(* CODESYS project BagFeeder.xml

Project tree, tasks and I/O mapping:
  function block BagFeeder [CFC]
*)

// BagFeeder
FUNCTION_BLOCK BagFeeder
//  .					.					.
VAR_INPUT
	BagOpenSensor: BOOL;
	IceFullSensor: BOOL;
	HeatSealOpened: BOOL;
	HeatSealClosed: BOOL;
	CheckBagOpenDelay: TIME;
	RetryBagOpenDelay: TIME;
	MaxIceFeedTime: TIME;
	IceTopOffTime: TIME;
	SealingTime: TIME;
	HeatSealCompleteDelay: TIME;
	//BagOpenRetries: UINT;
	
	BaggerSettings: BaggerSettings;
	
	Trigger: BOOL;
	MotionComplete: BOOL;
	
END_VAR
VAR_OUTPUT
	BlowerOn: BOOL;
	FillIce: BOOL;
	OpenHeatSeal: BOOL;
	CloseHeatSeal: BOOL;
	BagOpenRetryAttempts: UINT;
	
	ExecuteMotion: BOOL;
	MotionSteps: UDINT;
	MotionDirection: UINT;
	MotionSpeed: UINT;
	MotionTriggerOnSensor: BOOL;
END_VAR
VAR
	_MakeBagSequence: MakeBagSequence;
	_BagAdvanceSequence: BagAdvanceSequence; 
	_FeedIceSequence: FeedIceSequence;
	_SealBagSequence: SealBagSequence;
	
	_FailOpenCounter: CTU;
	_ResetFailCounter: BOOL;
	
	_MotionSelector: MotionSelector;
	
	_TestBagAdvance: BOOL;
	_TestFirstAdvance: BOOL;
	_TestFirstRetract: BOOL;
	_TestRetryAdvance: BOOL;
	_TestRetryRetract: BOOL;
	_TestTearBag: BOOL;
	_TestResetBag: BOOL;
	_TestRetractOneBag: BOOL;
	_TestBlowerOn: BOOL;
	MotionCompleteTrigger: R_TRIG;
	_TestHeatSeal: BOOL;
END_VAR
VAR // added by the converter: edge detectors and wires of the graphical bodies
    _w1, _w2, _w3, _w4, _w5, _w6, _w7, _w8 : ANY;
END_VAR

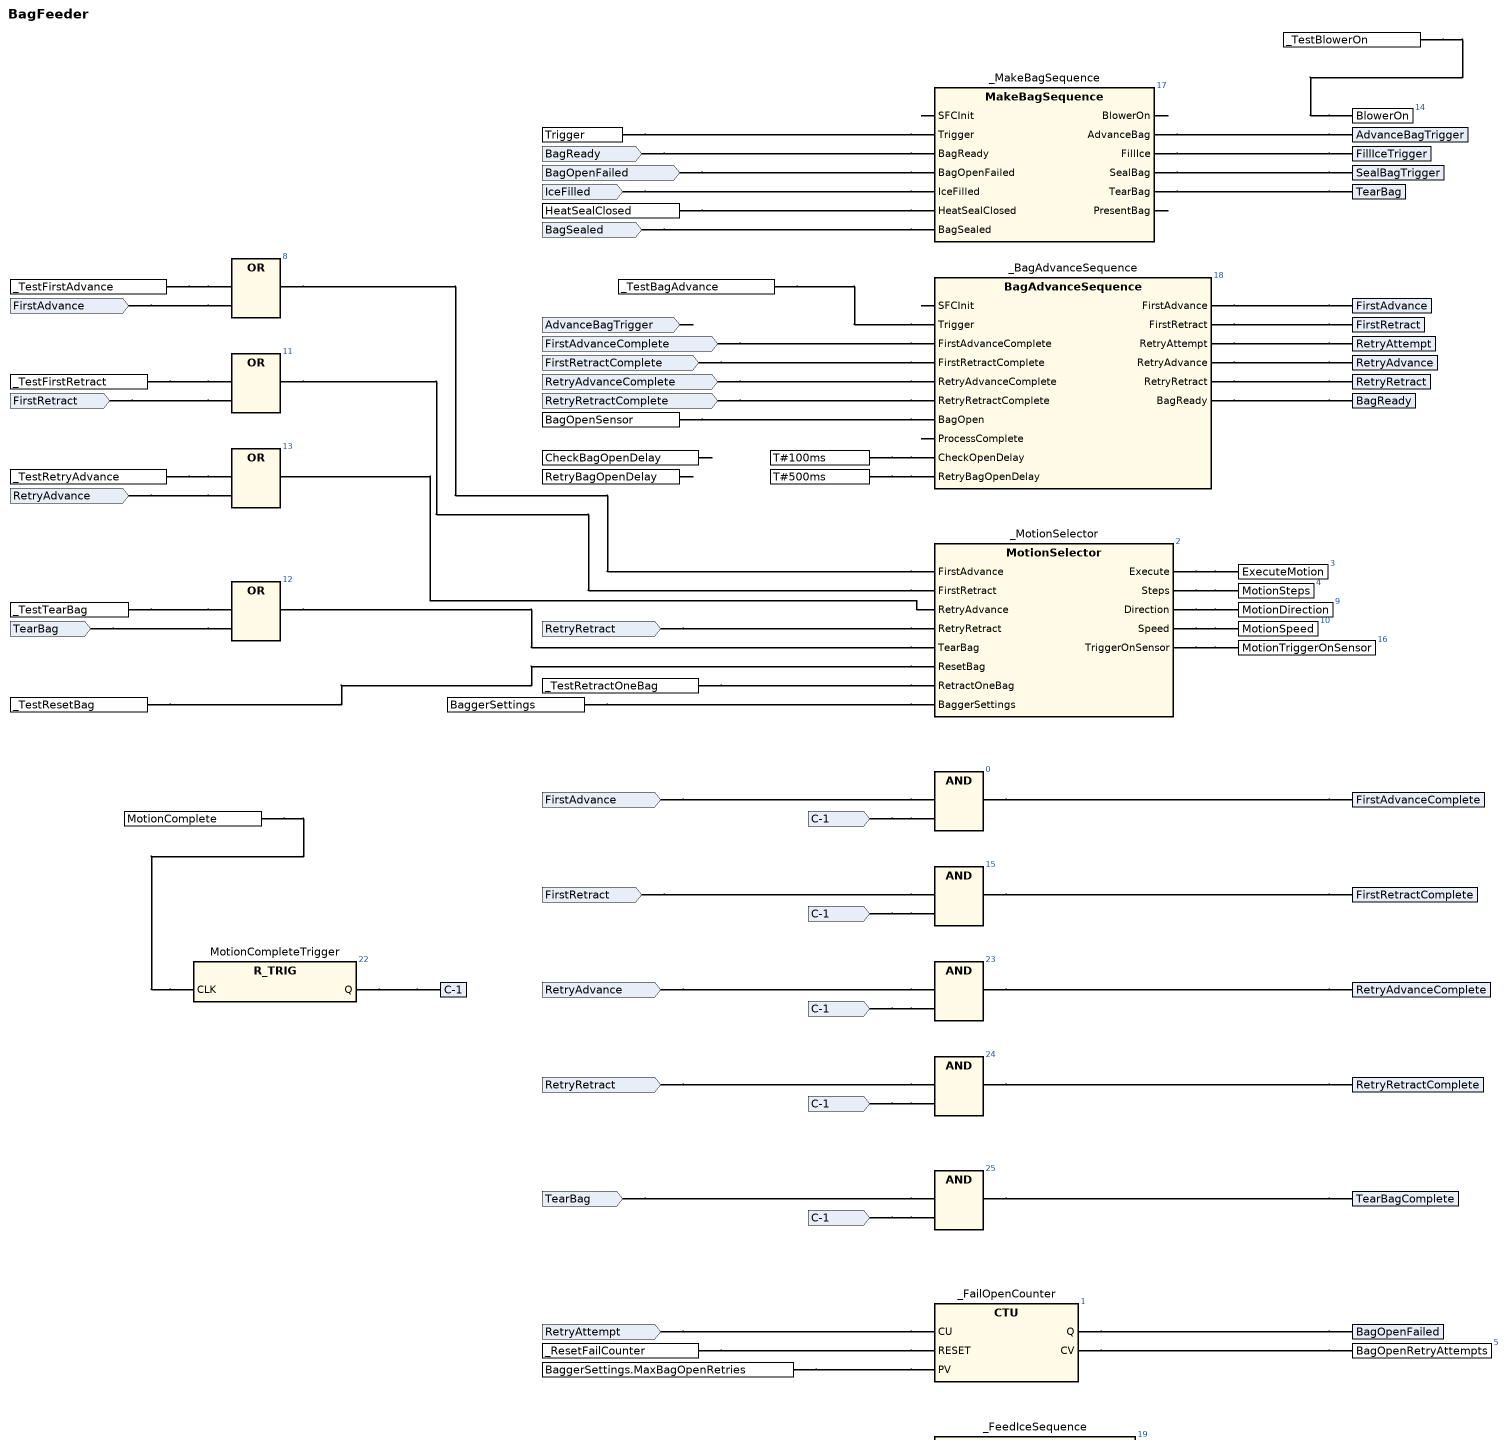
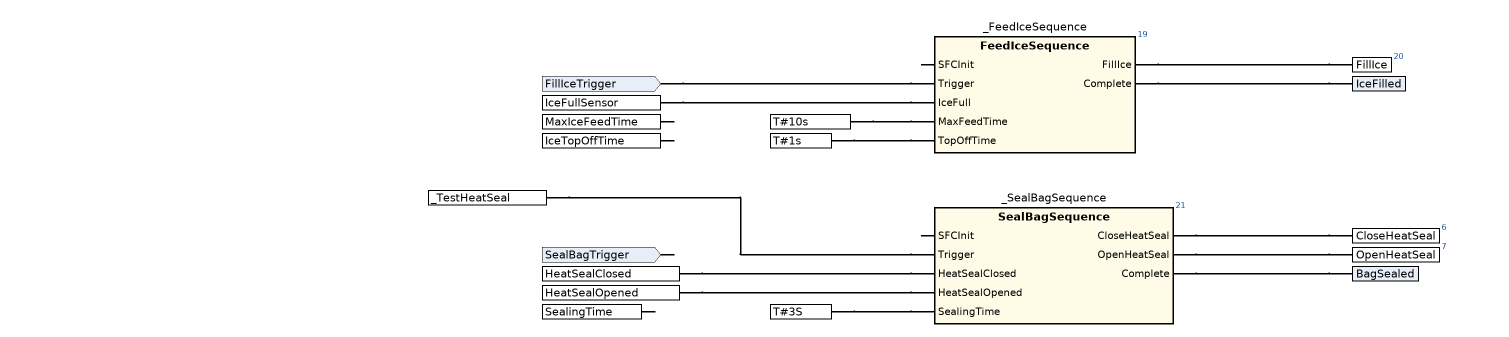
// note: 11 stored wires end on pins the file does not list and are not shown
_w1 := _BagAdvanceSequence.FirstAdvance AND MotionCompleteTrigger.Q;
_FailOpenCounter(
    CU := _BagAdvanceSequence.RetryAttempt,
    RESET := _ResetFailCounter,
    PV := BaggerSettings.MaxBagOpenRetries); // CTU
_MotionSelector(
    FirstAdvance := _w2,
    FirstRetract := _w3,
    RetryAdvance := _w4,
    RetryRetract := _BagAdvanceSequence.RetryRetract,
    TearBag := _w5,
    ResetBag := _TestResetBag,
    RetractOneBag := _TestRetractOneBag,
    BaggerSettings := BaggerSettings); // MotionSelector
ExecuteMotion := _MotionSelector.Execute;
MotionSteps := _MotionSelector.Steps;
BagOpenRetryAttempts := _FailOpenCounter.CV;
CloseHeatSeal := _SealBagSequence.CloseHeatSeal;
OpenHeatSeal := _SealBagSequence.OpenHeatSeal;
_w2 := _TestFirstAdvance OR _BagAdvanceSequence.FirstAdvance;
MotionDirection := _MotionSelector.Direction;
MotionSpeed := _MotionSelector.Speed;
_w3 := _TestFirstRetract OR _BagAdvanceSequence.FirstRetract;
_w5 := _TestTearBag OR _MakeBagSequence.TearBag;
_w4 := _TestRetryAdvance OR _BagAdvanceSequence.RetryAdvance;
BlowerOn := _TestBlowerOn;
_w6 := _BagAdvanceSequence.FirstRetract AND MotionCompleteTrigger.Q;
MotionTriggerOnSensor := _MotionSelector.TriggerOnSensor;
_MakeBagSequence(
    Trigger := Trigger,
    BagReady := _BagAdvanceSequence.BagReady,
    BagOpenFailed := _FailOpenCounter.Q,
    IceFilled := _FeedIceSequence.Complete,
    HeatSealClosed := HeatSealClosed,
    BagSealed := _SealBagSequence.Complete); // MakeBagSequence
_BagAdvanceSequence(
    Trigger := _TestBagAdvance,
    FirstAdvanceComplete := _w1,
    FirstRetractComplete := _w6,
    RetryAdvanceComplete := _w7,
    RetryRetractComplete := _w8,
    BagOpen := BagOpenSensor,
    CheckOpenDelay := T#100ms,
    RetryBagOpenDelay := T#500ms); // BagAdvanceSequence
_FeedIceSequence(
    Trigger := _MakeBagSequence.FillIce,
    IceFull := IceFullSensor,
    MaxFeedTime := T#10s,
    TopOffTime := T#1s); // FeedIceSequence
FillIce := _FeedIceSequence.FillIce;
_SealBagSequence(
    Trigger := _TestHeatSeal,
    HeatSealClosed := HeatSealClosed,
    HeatSealOpened := HeatSealOpened,
    SealingTime := T#3S); // SealBagSequence
MotionCompleteTrigger(CLK := MotionComplete); // R_TRIG
_w7 := _BagAdvanceSequence.RetryAdvance AND MotionCompleteTrigger.Q;
_w8 := _BagAdvanceSequence.RetryRetract AND MotionCompleteTrigger.Q;
(* _MakeBagSequence.TearBag AND MotionCompleteTrigger.Q; result not used *)
// CheckBagOpenDelay: input not connected
// RetryBagOpenDelay: input not connected
// MaxIceFeedTime: input not connected
// IceTopOffTime: input not connected
// SealingTime: input not connected

END_FUNCTION_BLOCK
